FUNCTION_BLOCK EA_network2
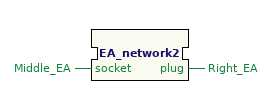
  SOCKETS
    socket : Middle_EA;
  END_SOCKETS
  PLUGS
    plug : Right_EA;
  END_PLUGS
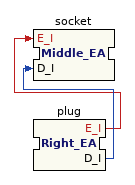
  EVENT_CONNECTIONS
    plug.E_I TO socket.E_I;
  END_CONNECTIONS
  DATA_CONNECTIONS
    plug.D_I TO socket.D_I;
  END_CONNECTIONS
END_FUNCTION_BLOCK
